{attribute 'Tc2GvlVarNames'}
{attribute 'strict'}
//Tipologia Ribaltino
TYPE e_Tipo_Ribaltino :
(
	RIBALTINO_NOT_DEFINED	:= -1,
	RIBALTINO_DOPO_SQUADRO  := 1, 		//Identifica il tipo di ribaltino diretto in linea, SENZA lo squadro
	RIBALTINO_DIRETTO 		:= 2 	//Identifica il tipo di ribaltino diretto in linea, SENZA lo squadro
);
END_TYPE
//  RIBALTINO_NOT_DEFINED = '-1'

(* stored: Version 1.1.0.1, ProductVersion 3.1.4024.11
   EnumerationTextList e_Tipo_Ribaltino: Id {e912fe23-7d52-4758-94a6-fe264bf31fb5} *)
